FUNCTION_BLOCK Conveyor_Belt_Model (* Basic Function Block Type *)
  (* Standard: 61499-2 *)
  (* Version 0.0, 2010-10-27, Gareth, nxtControl GmbH, Template *)
  (* Compiler header: package fb.rt.cs725; *)
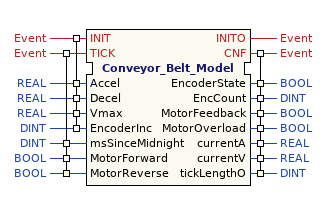
  EVENT_INPUT
    INIT WITH Accel, Decel, Vmax, EncoderInc; (* Initialization Request *)
    TICK WITH msSinceMidnight, MotorForward, MotorReverse; (* Normal Execution Request *)
  END_EVENT
  EVENT_OUTPUT
    INITO; (* Initialization Confirm *)
    CNF WITH EncoderState, EncCount, MotorFeedback, MotorOverload, currentA, currentV, tickLengthO; (* Execution Confirmation *)
  END_EVENT
  VAR_INPUT
    Accel : REAL;
    Decel : REAL;
    Vmax : REAL;
    EncoderInc : DINT;
    msSinceMidnight : DINT; (* Time in ms ULINT *)
    MotorForward : BOOL; (* ConveyorForward *)
    MotorReverse : BOOL; (* ConveyorReverse *)
  END_VAR
  VAR_OUTPUT
    EncoderState : BOOL; (* Output event qualifier *)
    EncCount : DINT;
    MotorFeedback : BOOL;
    MotorOverload : BOOL;
    currentA : REAL;
    currentV : REAL;
    tickLengthO : DINT;
  END_VAR
  VAR
    stopped : BOOL;
    LastStateChangeCount : DINT;
    count : DINT;
    msLastTick : DINT; (* LINT *)
    TickLength : DINT; (* Time elapsed in ms LINT *)
    V : REAL; (* Current velocity *)
    a : REAL; (* Current Acceleration / Decel *)
  END_VAR
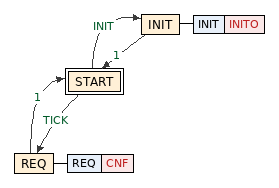
  EC_STATES
    START; (* Initial State *)
    INIT : INIT -> INITO; (* Initialization *)
    REQ : REQ -> CNF; (* Normal execution *)
  END_STATES
  EC_TRANSITIONS
    START TO INIT := INIT;
    INIT TO START := 1;
    START TO REQ := TICK;
    REQ TO START := 1;
  END_TRANSITIONS
  ALGORITHM INIT IN ST: (* Initialization algorithm *)
V := 0 ;
count := 0 ;
stopped := TRUE ;
  END_ALGORITHM
  ALGORITHM REQ IN ST: (* NB Acceleration removed Tick is called every 'instance of time' Times < 1x EncoderInc are unimportant Therefore a TICK == 1x EncoderInc ???   PASS // v && VMax are in mm PASS // EncoderInc is in (mm/10) printf("CBeltModel_TICK[%d] and \t\t\t\t\t%02x\n", me->ConvID, me->MotorStatus); *)
MotorFeedback := MotorForward;
//System.out.println("Motorforward = " + MotorForward);

// Accel and Decel are m/s/s, adjust for TickLength in ms *
IF msSinceMidnight >= msLastTick THEN
  TickLength := msSinceMidnight - msLastTick;
ELSE
  TickLength := 10000 + msSinceMidnight - msLastTick;
END_IF;
msLastTick := msSinceMidnight;

tickLengthO := TickLength;

IF MotorForward THEN
  stopped := FALSE;
  a := Accel * TickLength / 1000;
V:=Vmax;
// TODO: IF MotorReverse THEN
ELSE
  stopped := TRUE;
  a := -(Decel * TickLength / 1000);
  V:= 0;
END_IF;

currentA := a;
// a ~= Delta V

IF stopped THEN // Nothing to change
  RETURN;
END_IF;


 count := count + (V * TickLength);

IF ( V >= EncoderInc ) OR ( (count / EncoderInc) >  LastStateChangeCount ) THEN
  EncoderState := NOT EncoderState;
  LastStateChangeCount := (count / EncoderInc);
 END_IF;

EncCount := count;
  END_ALGORITHM
END_FUNCTION_BLOCK
